TYPE ST_VelocityConfig :
STRUCT
    fVelocity : LREAL;
END_STRUCT
END_TYPE

(* stored: Version 1.1.0.1, ProductVersion 3.1.4026.20
   DUT ST_VelocityConfig: Id {af5010a7-550e-47fd-9c91-445217d0a17f} *)
